// TIA Portal V15.1 export
// export: Created 2024-05-17T05:38:11.099427Z, ExportSetting WithDefaults, DisplayName Totally Integrated Automation Portal, DisplayVersion V15.1 Update 5, DisplayName TIA Portal Openness, DisplayVersion V15.1 Update 5, DisplayName SINAMICS Startdrive Advanced, DisplayVersion V15.1, DisplayName G130, G150, S120, S150, SINAMICS MV, S210, DisplayVersion V15.1, DisplayName G110M, G120, G120C, G120D, G120P, DisplayVersion V15.1, DisplayName STEP 7 Professional, DisplayVersion V15.1 Update 5, DisplayName STEP 7 Safety, DisplayVersion V15.1, DisplayName WinCC Professional, DisplayVersion V15.1 Update 5, DisplayName SIMATIC Visualization Architect, DisplayVersion V15.1
DATA_BLOCK "_PNDiagS7-1500_MAC"   // DB1012
{ S7_Optimized_Access := 'TRUE' }
VERSION : 0.1
// stored: AutoNumber false, DBAccessibleFromOPCUA true, InstanceOfName LPNIODiagMACS7-1500, InstanceOfType FB
"LPNIODiagMACS7-1500"
   // VAR_INPUT
   //    I_StartFillList { ExternalAccessible := 'False'; ExternalVisible := 'False'; ExternalWritable := 'False'} : Bool;
   //    I_LastDeviceNumber { ExternalAccessible := 'False'; ExternalVisible := 'False'; ExternalWritable := 'False'} : Int;
   // END_VAR
   // VAR_OUTPUT
   //    O_Done { ExternalAccessible := 'False'; ExternalVisible := 'False'; ExternalWritable := 'False'} : Bool;
   //    O_MACAddress { ExternalAccessible := 'False'; ExternalVisible := 'False'; ExternalWritable := 'False'} : Array[0..255] of String[18];
   // END_VAR
   // VAR_IN_OUT
   //    IO_DeviceExist : Array[0..255] of Bool;
   //    IO_HWIdentifier : Array[0..255] of UInt;
   //    IO_GetStationMAC : Array[0..255] of IF_CONF_MAC;
   // END_VAR
   // VAR
   //    Index { ExternalAccessible := 'False'; ExternalVisible := 'False'; ExternalWritable := 'False'} : Int;
   //    LastDeviceNumber { ExternalAccessible := 'False'; ExternalVisible := 'False'; ExternalWritable := 'False'} : Int;
   //    Done { ExternalAccessible := 'False'; ExternalVisible := 'False'; ExternalWritable := 'False'} : Bool;
   //    DoneDelay { ExternalAccessible := 'False'; ExternalVisible := 'False'; ExternalWritable := 'False'} : Bool;
   //    ReturnGetStationInfoBusy_MAC { ExternalAccessible := 'False'; ExternalVisible := 'False'; ExternalWritable := 'False'} : Bool;
   //    ReturnGetStationInfoDone_MAC { ExternalAccessible := 'False'; ExternalVisible := 'False'; ExternalWritable := 'False'} : Bool;
   //    ReturnGetStationInfoError_MAC { ExternalAccessible := 'False'; ExternalVisible := 'False'; ExternalWritable := 'False'} : Bool;
   //    ReturnGetStationInfoStatus_MAC { ExternalAccessible := 'False'; ExternalVisible := 'False'; ExternalWritable := 'False'} : Word;
   //    MACAddress_ADDR1 { ExternalAccessible := 'False'; ExternalVisible := 'False'; ExternalWritable := 'False'} : String[2];
   //    MACAddress_ADDR2 { ExternalAccessible := 'False'; ExternalVisible := 'False'; ExternalWritable := 'False'} : String[2];
   //    MACAddress_ADDR3 { ExternalAccessible := 'False'; ExternalVisible := 'False'; ExternalWritable := 'False'} : String[2];
   //    MACAddress_ADDR4 { ExternalAccessible := 'False'; ExternalVisible := 'False'; ExternalWritable := 'False'} : String[2];
   //    MACAddress_ADDR5 { ExternalAccessible := 'False'; ExternalVisible := 'False'; ExternalWritable := 'False'} : String[2];
   //    MACAddress_ADDR6 { ExternalAccessible := 'False'; ExternalVisible := 'False'; ExternalWritable := 'False'} : String[2];
   //    MACAddress { ExternalAccessible := 'False'; ExternalVisible := 'False'; ExternalWritable := 'False'} : String[18];
   //    RetVal { ExternalAccessible := 'False'; ExternalVisible := 'False'; ExternalWritable := 'False'} : Word;
   //    GetStationInfo_MAC { ExternalAccessible := 'False'; ExternalVisible := 'False'; ExternalWritable := 'False'; S7_SetPoint := 'True'} : GetStationInfo;
   //    TimerDone { ExternalAccessible := 'False'; ExternalVisible := 'False'; ExternalWritable := 'False'; S7_SetPoint := 'True'} : TON_TIME;
   //    EdgeStartFillList { ExternalAccessible := 'False'; ExternalVisible := 'False'; ExternalWritable := 'False'; S7_SetPoint := 'True'} : R_TRIG;
   // END_VAR
BEGIN
END_DATA_BLOCK
